INTERFACE ITcoDoorLock

{attribute 'monitoring' := 'call'}
PROPERTY IsClosed : BOOL
GET
END_GET
END_PROPERTY

{attribute 'monitoring' := 'call'}
PROPERTY IsLocked : BOOL
GET
END_GET
END_PROPERTY

{attribute 'monitoring' := 'call'}
PROPERTY IsOpen : BOOL
GET
END_GET
END_PROPERTY

METHOD Lock : BOOL
VAR_INPUT
END_VAR
END_METHOD

METHOD UnLock : BOOL
VAR_INPUT
END_VAR
END_METHOD

END_INTERFACE

(* stored: Version 1.1.0.1
   Itf ITcoDoorLock: Id {e31e81a9-23a6-4ec0-a9de-53d13304f8f9}
   Property IsClosed: Id {dc58be1e-9932-4bc5-a4c3-9c5de040df19}
   Get Get: Id {28afa32b-63f2-493f-b6df-d1731d233750}
   Property IsLocked: Id {86c0bd4f-8a0a-493e-9e37-4af93e1720f7}
   Get Get: Id {51f88c03-2ce8-43e1-a901-bc1e5866bb3b}
   Property IsOpen: Id {2872ec8e-80c0-420a-af22-60ff31cc645a}
   Get Get: Id {29fb5cc9-a453-4b32-8c00-a5e4e461d0da}
   Method Lock: Id {de9819e3-e479-47e4-86b1-0481c1da514b}
   Method UnLock: Id {9671c65f-e54a-4699-b621-54671fc3df5a} *)
